INTERFACE I_BacklashCompensation EXTENDS I_Error

METHOD BacklashCompensation
VAR_INPUT
	Enable : BOOL := FALSE;
	RampVelo : LREAL;
END_VAR
END_METHOD

PROPERTY Busy : BOOL
GET
END_GET
END_PROPERTY

PROPERTY CurrentBacklash : LREAL
GET
END_GET
END_PROPERTY

METHOD EnableBacklashCompensation
VAR_INPUT
    UserEnable : BOOL;
    Compensation : LREAL;
END_VAR
END_METHOD

PROPERTY Status : BOOL
GET
END_GET
END_PROPERTY

END_INTERFACE

(* stored: Version 1.1.0.1
   Itf I_BacklashCompensation: Id {c0dc76c5-ea53-4a27-aade-dbf12ab6b44d}
   Method BacklashCompensation: Id {3665b988-9224-4240-a54c-db8e420c5cde}
   Property Busy: Id {e81610e6-4246-42a9-939b-3c713737277b}
   Get Get: Id {38e42d74-d048-4efa-9d44-c00553c24d88}
   Property CurrentBacklash: Id {ff081112-3182-493d-846e-c2192c5f77d6}
   Get Get: Id {5dbd065d-c6db-421a-8993-7aa4f3a00024}
   Method EnableBacklashCompensation: Id {e97f2fd7-00e3-4003-9a19-7946698414f6}
   Property Status: Id {dd023d24-4958-4a64-8af6-f09a6b1978e9}
   Get Get: Id {2244ed4b-ffad-4d7c-8cbb-2047985c42a1} *)
